FUNCTION_BLOCK ServoNC EXTENDS FBA_TrifectaDrive IMPLEMENTS I_EncodedDrive
VAR_OUTPUT	
	ready : BOOL;
	position : LREAL;
	velocity : LREAL;
END_VAR
VAR
	axis : AXIS_REF;
	
	mcReadPosition : MC_ReadActualPosition;
	mcReadVelocity : MC_ReadActualVelocity;
	mcReadError : MC_ReadAxisError;
	mcReset : MC_Reset;
	
	mcPower : MC_Power;
	mcMoveAbsolute : MC_MoveAbsolute;
	mcMoveRelative : MC_MoveRelative;
	mcMoveVelocity : MC_MoveVelocity;
	
	mcSetPosition : MC_SetPosition;
	mcStop : MC_Stop;
END_VAR
VAR_STAT CONSTANT
	targetingVelocity : INT := 500;
	continuousVelocity : INT := 100;
END_VAR

override();

blocks();

mcReset.Execute := FALSE;
mcMoveAbsolute.Execute := FALSE;
mcMoveRelative.Execute := FALSE;
mcMoveVelocity.Execute := FALSE;
mcSetPosition.Execute := FALSE;
mcStop.Execute := FALSE;

blocks();

ready := bEnable AND NOT Active AND HomeSet;

PROPERTY Active : BOOL
GET
Active := 
	mcMoveAbsolute.Busy OR 
	mcMoveRelative.Busy OR 
	mcMoveVelocity.Busy OR 
	mcSetPosition.Busy OR 
	mcReset.Busy OR 
	mcStop.Busy OR 
	step <> 0;
END_GET
END_PROPERTY

METHOD PRIVATE blocks : BOOL
mcReadPosition(
	Axis:= axis, 
	Enable:= TRUE, 
	Valid=> , 
	Busy=> , 
	Error=> , 
	ErrorID=> , 
	Position=> position);
	
mcReadVelocity(
	Axis:= axis, 
	Enable:= TRUE, 
	Valid=> , 
	Busy=> , 
	Error=> , 
	ErrorID=> , 
	ActualVelocity=> velocity);
	
mcReadError(
	Axis:= axis, 
	Enable:= TRUE, 
	Valid=> , 
	Busy=> , 
	Error=> , 
	ErrorID=> , 
	AxisErrorID=> );

mcReset(
	Axis:= axis, 
	Execute:= , 
	Done=> , 
	Busy=> , 
	Error=> , 
	ErrorID=> );

mcPower(
	Axis:= axis, 
	Enable:= bEnable, 
	Enable_Positive:= TRUE, 
	Enable_Negative:= TRUE, 
	Override:= 100, 
	BufferMode:= , 
	Options:= , 
	Status=> , 
	Busy=> , 
	Active=> , 
	Error=> , 
	ErrorID=> );

mcMoveAbsolute(
	Axis:= axis, 
	Execute:= , 
	Position:= , 
	Velocity:= targetingVelocity, 
	Acceleration:= , 
	Deceleration:= , 
	Jerk:= , 
	BufferMode:= , 
	Options:= , 
	Done=> , 
	Busy=> , 
	Active=> , 
	CommandAborted=> , 
	Error=> , 
	ErrorID=> );
	
mcMoveRelative(
	Axis:= axis, 
	Execute:= , 
	Distance:= ,
	Velocity:= targetingVelocity, 
	Acceleration:= , 
	Deceleration:= , 
	Jerk:= , 
	BufferMode:= , 
	Options:= , 
	Done=> , 
	Busy=> , 
	Active=> , 
	CommandAborted=> , 
	Error=> , 
	ErrorID=> );
	
mcMoveVelocity( //stopped with stop();
	Axis:= axis, 
	Execute:= , 
	Velocity:= continuousVelocity, 
	Acceleration:= , 
	Deceleration:= , 
	Jerk:= , 
	Direction:= , 
	BufferMode:= , 
	Options:= , 
	InVelocity=> , 
	Busy=> , 
	Active=> , 
	CommandAborted=> , 
	Error=> , 
	ErrorID=> );
	
mcSetPosition(
	Axis:= axis, 
	Execute:= , 
	Position:= , 
	Mode:= , 
	Options:= , 
	Done=> , 
	Busy=> , 
	Error=> , 
	ErrorID=> );
	
mcStop(
	Axis:= axis, 
	Execute:= , 
	Deceleration:= , 
	Jerk:= , 
	Options:= , 
	Done=> , 
	Busy=> , 
	Active=> , 
	CommandAborted=> , 
	Error=> , 
	ErrorID=> );
END_METHOD

PROPERTY CurrentPosition : LREAL
GET
CurrentPosition := position;
END_GET
SET
position := CurrentPosition;
END_SET
END_PROPERTY

PROPERTY Error : BOOL
GET
error := 
	mcMoveAbsolute.Error OR 
	mcMoveRelative.Error OR 
	mcMoveVelocity.Error OR 
	mcSetPosition.Error OR 
	mcReset.Error OR 
	mcStop.Error OR
	mcReadError.AxisErrorID > 0;
END_GET
END_PROPERTY

METHOD homingSequence : BOOL
CASE step OF
	Homing.IDLE:
		reset();
		IF bEnable THEN
			step := Homing.START;
		END_IF
		
	Homing.START:
		IF AtHome THEN
			mcMoveVelocity.Execute := FALSE;
			step := Homing.STOP;
			
		ELSIF AtInnerLimit THEN
			mcMoveVelocity.Execute := FALSE;
			step := Homing.RETRY;
			
		ELSE
			mcMoveVelocity.Direction := MC_Negative_Direction;
			mcMoveVelocity.Execute := NOT mcMoveVelocity.Execute;
		END_IF
		
	Homing.RETRY:
		IF AtOuterLimit THEN
			mcMoveVelocity.Execute := FALSE;
			step := Homing.START;
		ELSE
			mcMoveVelocity.Direction := MC_Positive_Direction;
			mcMoveVelocity.Execute := NOT mcMoveVelocity.Execute;
		END_IF
		
	Homing.STOP:
		IF velocity = 0 THEN
			mcStop.Execute := FALSE;
			step := Homing.SET;
		ELSE
			mcStop.Execute := TRUE;
		END_IF
		
	Homing.SET:
		IF position = 0 THEN
			mcSetPosition.Execute := FALSE;
			homingSequence := TRUE;
			step := Homing.DONE;
		ELSE
			mcSetPosition.Position := 0;
			mcSetPosition.Execute := TRUE;
		END_IF
		
	Homing.DONE:
		homingComplete := TRUE;
		step := Homing.IDLE;
		
END_CASE
END_METHOD

METHOD moveAbsolute : BOOL
VAR_INPUT
	newTarget : LREAL;
END_VAR
(*
VAR_OUTPUT
	fault : BOOL;
END_VAR
*)
IF NOT Active AND NOT error THEN
	mcMoveAbsolute.Position := newTarget;
	mcMoveAbsolute.Execute := TRUE;
END_IF

moveAbsolute := (*mcMoveAbsolute.Done AND mcMoveAbsolute.Active;*)
	position = newTarget;
END_METHOD

METHOD moveContinuous : BOOL
VAR_INPUT
	//direction : BOOL; //direction (F = inwards, T = outwards)
	direction : MC_Direction;
END_VAR
(*
IF mcMoveVelocity.Active THEN
	stop();
END_IF

IF NOT mcStop.Done THEN
	RETURN;
END_IF
*)
(*
IF direction THEN
	mcMoveVelocity.Direction := MC_Positive_Direction;
ELSE
	mcMoveVelocity.Direction := MC_Negative_Direction;
END_IF
*)
mcMoveVelocity.Direction := direction;

IF NOT mcMoveVelocity.Error THEN
	mcMoveVelocity.Execute := TRUE;
	moveContinuous := TRUE;
END_IF
END_METHOD

METHOD moveRelative : BOOL
VAR_INPUT
	distance : LREAL;
END_VAR
mcMoveRelative.Distance := distance;

moveRelative := mcMoveRelative.Done;
END_METHOD

METHOD PRIVATE override : BOOL
VAR_INPUT
END_VAR
(*
-at home and attempting to traverse outward
-at outer limit and attempting to traverse outward
-at inner limit and attempting to traverse inwards
*)
(*
inward = negative direction, negative velocity
outward = positive direction, positive velocity
*)

IF error THEN
	stop();
	reset();
	
ELSIF
	AtHome AND (TargetPosition > CurrentPosition OR velocity > 0) OR
	AtInnerLimit AND (TargetPosition > CurrentPosition OR velocity > 0) OR
	AtOuterLimit AND (TargetPosition < CurrentPosition OR velocity < 0)
THEN
	stop();
END_IF
END_METHOD

METHOD reset : BOOL
VAR_INPUT
END_VAR
mcReset.Execute := TRUE;

reset := mcReset.Done;
END_METHOD

METHOD stop : BOOL
VAR_INPUT
END_VAR
mcStop.Execute := TRUE;

mcMoveAbsolute.Execute := FALSE;
mcMoveRelative.Execute := FALSE;
mcMoveVelocity.Execute := FALSE;
END_METHOD

PROPERTY TargetPosition : LREAL
GET
END_GET
SET
moveAbsolute(newTarget := TargetPosition);
END_SET
END_PROPERTY

METHOD toHome : BOOL
VAR_INPUT
END_VAR
moveAbsolute(newTarget := 0);

toHome := AtHome;
END_METHOD

END_FUNCTION_BLOCK

(* stored: Version 1.1.0.1, ProductVersion 3.1.4024.11
   POU ServoNC: Id {32a5f031-8d9d-4fd1-beaa-c11419499820}, SpecialFunc None
   Folder Private: Id {33b8f8d7-2454-4b48-8826-e669a7a71373}
   Folder Properties: Id {de97ab30-a5ce-41f8-9a7f-899063ea2e89}
   Property Active: Id {9a2dc098-5061-43cc-b878-8a169e02b216}
   Get Get: Id {91a772c4-68a7-43be-946c-4606b5409550}
   Method blocks: Id {8e7ecd71-b8e2-494e-8f60-f755d355f9cb}
   Property CurrentPosition: Id {2badad16-95ce-48ed-aaee-135b30279ac7}
   Get Get: Id {f756b0a1-2c58-48d0-a153-2df584dee434}
   Set Set: Id {d2e54576-8dbc-4206-86cb-001891f8afe5}
   Property Error: Id {465d2e0f-de23-4c71-8c88-204b9a266cb7}
   Get Get: Id {17c06e5f-a35d-4019-a4ac-edc4030e0a39}
   Method homingSequence: Id {aecbd1e9-e22a-4ed3-a925-c3231352561d}
   Method moveAbsolute: Id {3f975309-5c53-405d-9f0b-e579b06b055e}
   Method moveContinuous: Id {478a39e7-1e41-4b59-bc73-67d5f0d90925}
   Method moveRelative: Id {12c4833e-0589-4eeb-977e-183fc7b9d136}
   Method override: Id {79dc4e8a-f0f6-429c-85fb-2ad70e9ac6ef}
   Method reset: Id {eb325f3d-ea87-4834-94f6-db83f102b678}
   Method stop: Id {51177749-aac1-491b-bfc8-5908f17a143a}
   Property TargetPosition: Id {9b616396-095b-4580-9a0a-bb8838fb03a9}
   Get Get: Id {cd7a3365-f676-4cbd-b8d7-59559079d95b}
   Set Set: Id {54a62271-53ac-4ce8-8bd9-e38bce043066}
   Method toHome: Id {0f624974-229f-4b55-9e8d-00320dad6eb5} *)
